VAR_GLOBAL
	fJoyX : LREAL;
	fJoyY : LREAL;
END_VAR

(* stored: Version 1.1.0.1, ProductVersion 3.1.4024.12
   GVL G_Inputs: Id {1b387283-05cb-4799-bd28-84ac7ae3617c} *)
